Staubli VAL3: IO.dtx

public aio aAio{}
  [In4_a7CurPosH] = {link=ModbusSrv-0\Modbus-Word\In4_a7CurPosH}
  [In4_a7CurPosL] = {link=ModbusSrv-0\Modbus-Word\In4_a7CurPosL}
  [In4_a8CurPosH] = {link=ModbusSrv-0\Modbus-Word\In4_a8CurPosH}
  [In4_a8CurPosL] = {link=ModbusSrv-0\Modbus-Word\In4_a8CurPosL}
  [In_aVersion] = {link=ModbusSrv-0\Modbus-Word\In_aVersion}
  [O1_aAirPress] = {link=ModbusSrv-0\Modbus-Word\O1_aAirPress}
  [O1_aFPWM] = {link=ModbusSrv-0\Modbus-Word\O1_aFPWM}
  [O1_aLasPwr] = {link=ModbusSrv-0\Modbus-Word\O1_aLasPwr}
  [O1_aPMW] = {link=ModbusSrv-0\Modbus-Word\O1_aPMW}
  [O2_aFollowSensitive] = {link=ModbusSrv-0\Modbus-Word\O2_aFollowSensitive}
  [O2_aNull] = {link=ModbusSrv-0\Modbus-Word\O2_aNull}
  [O4_a7AiHomeH] = {link=ModbusSrv-0\Modbus-Word\O4_a7AiHomeH}
  [O4_a7AiHomeL] = {link=ModbusSrv-0\Modbus-Word\O4_a7AiHomeL}
  [O4_a7JogVelo] = {link=ModbusSrv-0\Modbus-Word\O4_a7JogVelo}
  [O4_a7MoveDis] = {link=ModbusSrv-0\Modbus-Word\O4_a7MoveDis}
  [O4_a7MovePosH] = {link=ModbusSrv-0\Modbus-Word\O4_a7MovePosH}
  [O4_a7MovePosL] = {link=ModbusSrv-0\Modbus-Word\O4_a7MovePosL}
  [O4_a7Velocity] = {link=ModbusSrv-0\Modbus-Word\O4_a7Velocity}
  [O4_a8AiHomeH] = {link=ModbusSrv-0\Modbus-Word\O4_a8AiHomeH}
  [O4_a8AiHomeL] = {link=ModbusSrv-0\Modbus-Word\O4_a8AiHomeL}
  [O4_a8JogVelo] = {link=ModbusSrv-0\Modbus-Word\O4_a8JogVelo}
  [O4_a8MoveDis] = {link=ModbusSrv-0\Modbus-Word\O4_a8MoveDis}
  [O4_a8MovePosH] = {link=ModbusSrv-0\Modbus-Word\O4_a8MovePosH}
  [O4_a8MovePosL] = {link=ModbusSrv-0\Modbus-Word\O4_a8MovePosL}
  [O4_a8Velocity] = {link=ModbusSrv-0\Modbus-Word\O4_a8Velocity}
  [Out_a114_129] = {link=ModbusSrv-0\Modbus-Word\Out_a114_129}
  [Out_a130_133] = {link=ModbusSrv-0\Modbus-Word\Out_a130_133}
  [Out_a66_81] = {link=ModbusSrv-0\Modbus-Word\Out_a66_81}
  [Out_a82_97] = {link=ModbusSrv-0\Modbus-Word\Out_a82_97}
  [Out_a98_113] = {link=ModbusSrv-0\Modbus-Word\Out_a98_113}
public bool bAxisDoorEnable
bool bDigFollowHight
public bool bDigtal[167]
  [0] = true
  [1] = true
  [2] = true
  [3] = true
  [4] = true
  [5] = true
  [6] = true
  [7] = true
  [8] = true
  [9] = true
  [10] = true
  [11] = true
  [12] = true
  [13] = true
  [14] = true
  [15] = true
  [16] = true
  [17] = true
  [18] = true
  [19] = true
  [20] = true
  [21] = true
  [22] = true
  [23] = true
  [24] = true
  [25] = true
  [26] = true
  [27] = true
  [28] = true
  [29] = true
  [30] = true
  [31] = true
  [32] = true
  [33] = true
  [34] = true
  [35] = true
  [36] = true
  [37] = true
  [38] = true
  [39] = true
  [40] = true
  [41] = true
  [42] = true
  [43] = true
  [44] = true
  [45] = true
  [46] = true
  [47] = true
  [48] = true
  [49] = true
  [50] = true
  [51] = true
  [52] = true
  [53] = true
  [54] = true
  [55] = true
  [56] = true
  [57] = true
  [58] = true
  [59] = true
  [60] = true
  [61] = true
  [62] = true
  [63] = true
  [64] = true
  [65] = true
  [66] = true
  [67] = true
  [68] = true
  [69] = true
  [70] = true
  [71] = true
  [72] = true
  [73] = true
  [74] = true
  [75] = true
  [76] = true
  [77] = true
  [78] = true
  [79] = true
  [80] = true
  [81] = true
  [82] = true
  [83] = true
  [84] = true
  [85] = true
  [86] = true
  [87] = true
  [88] = true
  [89] = true
  [90] = true
  [91] = true
  [92] = true
  [93] = true
  [94] = true
  [95] = true
  [96] = true
  [97] = true
  [98] = true
  [99] = true
  [100] = true
  [101] = true
  [102] = true
  [103] = true
  [104] = true
  [105] = true
  [106] = true
  [107] = true
  [108] = true
  [109] = true
  [110] = true
  [111] = true
  [112] = true
  [113] = true
  [114] = true
  [115] = true
  [116] = true
  [117] = true
  [118] = true
  [119] = true
  [120] = true
  [121] = true
  [122] = true
  [123] = true
  [124] = true
  [125] = true
  [126] = true
  [127] = true
  [128] = true
  [129] = true
  [130] = true
  [131] = true
  [132] = true
  [133] = true
  [134] = true
public bool bExt7AxisEnable
public bool bExt8AxisEnable
public bool bGunUp
bool bWaitActionOff
bool bWaitFollowDown
public bool bWeldEnable
public dio dDio{}
  [In1_bEndCycl] = {link=ModbusSrv-0\Modbus-Bit\In1_bEndCycl}
  [In1_bHome] = {link=ModbusSrv-0\Modbus-Bit\In1_bHome}
  [In1_bNull1] = {link=ModbusSrv-0\Modbus-Bit\In1_bNull1}
  [In1_bNull2] = {link=ModbusSrv-0\Modbus-Bit\In1_bNull2}
  [In1_bNull3] = {link=ModbusSrv-0\Modbus-Bit\In1_bNull3}
  [In1_bOutAlarm] = {link=ModbusSrv-0\Modbus-Bit\In1_bOutAlarm}
  [In1_bPausCycl] = {link=ModbusSrv-0\Modbus-Bit\In1_bPausCycl}
  [In1_bPeripheralReady] = {link=ModbusSrv-0\Modbus-Bit\In1_bPeripheralReady}
  [In1_bPowerOn] = {link=ModbusSrv-0\Modbus-Bit\In1_bPowerOn}
  [In1_bPrdSta1] = {link=ModbusSrv-0\Modbus-Bit\In1_bPrdSta1}
  [In1_bPrdSta2] = {link=ModbusSrv-0\Modbus-Bit\In1_bPrdSta2}
  [In1_bReset] = {link=ModbusSrv-0\Modbus-Bit\In1_bReset}
  [In1_bStartCycl] = {link=ModbusSrv-0\Modbus-Bit\In1_bStartCycl}
  [In1_bStopCycl] = {link=ModbusSrv-0\Modbus-Bit\In1_bStopCycl}
  [In2_bAirAlarm] = {link=ModbusSrv-0\Modbus-Bit\In2_bAirAlarm}
  [In2_bCollisonAlarm] = {link=ModbusSrv-0\Modbus-Bit\In2_bCollisonAlarm}
  [In2_bContactAlarm] = {link=ModbusSrv-0\Modbus-Bit\In2_bContactAlarm}
  [In2_bLaserAlarm] = {link=ModbusSrv-0\Modbus-Bit\In2_bLaserAlarm}
  [In2_bNull1] = {link=ModbusSrv-0\Modbus-Bit\In2_bNull1}
  [In2_bNull2] = {link=ModbusSrv-0\Modbus-Bit\In2_bNull2}
  [In2_bNull3] = {link=ModbusSrv-0\Modbus-Bit\In2_bNull3}
  [In2_bNull4] = {link=ModbusSrv-0\Modbus-Bit\In2_bNull4}
  [In2_bNull5] = {link=ModbusSrv-0\Modbus-Bit\In2_bNull5}
  [In2_bNull6] = {link=ModbusSrv-0\Modbus-Bit\In2_bNull6}
  [In2_bNull7] = {link=ModbusSrv-0\Modbus-Bit\In2_bNull7}
  [In2_bNull8] = {link=ModbusSrv-0\Modbus-Bit\In2_bNull8}
  [In2_bNull9] = {link=ModbusSrv-0\Modbus-Bit\In2_bNull9}
  [In2_bPrdSta3] = {link=ModbusSrv-0\Modbus-Bit\In2_bPrdSta3}
  [In2_bPrdSta4] = {link=ModbusSrv-0\Modbus-Bit\In2_bPrdSta4}
  [In2_bRasterOn] = {link=ModbusSrv-0\Modbus-Bit\In2_bRasterOn}
  [In4_b7BackHome] = {link=ModbusSrv-0\Modbus-Bit\In4_b7BackHome}
  [In4_b7HomeDone] = {link=ModbusSrv-0\Modbus-Bit\In4_b7HomeDone}
  [In4_b7IsHome] = {link=ModbusSrv-0\Modbus-Bit\In4_b7IsHome}
  [In4_b7MotorError] = {link=ModbusSrv-0\Modbus-Bit\In4_b7MotorError}
  [In4_b7MotorPower] = {link=ModbusSrv-0\Modbus-Bit\In4_b7MotorPower}
  [In4_b7Reached] = {link=ModbusSrv-0\Modbus-Bit\In4_b7Reached}
  [In4_b8BackHome] = {link=ModbusSrv-0\Modbus-Bit\In4_b8BackHome}
  [In4_b8HomeDone] = {link=ModbusSrv-0\Modbus-Bit\In4_b8HomeDone}
  [In4_b8IsHome] = {link=ModbusSrv-0\Modbus-Bit\In4_b8IsHome}
  [In4_b8MotorError] = {link=ModbusSrv-0\Modbus-Bit\In4_b8MotorError}
  [In4_b8MotorPower] = {link=ModbusSrv-0\Modbus-Bit\In4_b8MotorPower}
  [In4_b8Reached] = {link=ModbusSrv-0\Modbus-Bit\In4_b8Reached}
  [In4_bNull1] = {link=ModbusSrv-0\Modbus-Bit\In4_bNull1}
  [In4_bNull2] = {link=ModbusSrv-0\Modbus-Bit\In4_bNull2}
  [In4_bNull3] = {link=ModbusSrv-0\Modbus-Bit\In4_bNull3}
  [In4_bNull4] = {link=ModbusSrv-0\Modbus-Bit\In4_bNull4}
  [In4_bNull5] = {link=ModbusSrv-0\Modbus-Bit\In4_bNull5}
  [In4_bNull6] = {link=ModbusSrv-0\Modbus-Bit\In4_bNull6}
  [In4_bNull7] = {link=ModbusSrv-0\Modbus-Bit\In4_bNull7}
  [In4_bNull8] = {link=ModbusSrv-0\Modbus-Bit\In4_bNull8}
  [In7_bDownLimit_7] = {link=ModbusSrv-0\Modbus-Bit\In7_bDownLimit_7}
  [In7_bHomeLimit_7] = {link=ModbusSrv-0\Modbus-Bit\In7_bHomeLimit_7}
  [In7_bNull1] = {link=ModbusSrv-0\Modbus-Bit\In7_bNull1}
  [In7_bUpLimit_7] = {link=ModbusSrv-0\Modbus-Bit\In7_bUpLimit_7}
  [In8_bDownLimit_8] = {link=ModbusSrv-0\Modbus-Bit\In8_bDownLimit_8}
  [In8_bHomeLimit_8] = {link=ModbusSrv-0\Modbus-Bit\In8_bHomeLimit_8}
  [In8_bNull1] = {link=ModbusSrv-0\Modbus-Bit\In8_bNull1}
  [In8_bUpLimit_8] = {link=ModbusSrv-0\Modbus-Bit\In8_bUpLimit_8}
  [O1_bAirOn] = {link=ModbusSrv-0\Modbus-Bit\O1_bAirOn}
  [O1_bAlarm] = {link=ModbusSrv-0\Modbus-Bit\O1_bAlarm}
  [O1_bFollowDone] = {link=ModbusSrv-0\Modbus-Bit\O1_bFollowDone}
  [O1_bFollowOn] = {link=ModbusSrv-0\Modbus-Bit\O1_bFollowOn}
  [O1_bGreenLamp] = {link=ModbusSrv-0\Modbus-Bit\O1_bGreenLamp}
  [O1_bLaserOn] = {link=ModbusSrv-0\Modbus-Bit\O1_bLaserOn}
  [O1_bNull1] = {link=ModbusSrv-0\Modbus-Bit\O1_bNull1}
  [O1_bRedLamp] = {link=ModbusSrv-0\Modbus-Bit\O1_bRedLamp}
  [O1_bYellowLamp] = {link=ModbusSrv-0\Modbus-Bit\O1_bYellowLamp}
  [O2_bAxisPos1] = {link=ModbusSrv-0\Modbus-Bit\O2_bAxisPos1}
  [O2_bAxisPos2] = {link=ModbusSrv-0\Modbus-Bit\O2_bAxisPos2}
  [O2_bAxisPos3] = {link=ModbusSrv-0\Modbus-Bit\O2_bAxisPos3}
  [O2_bFollowHeigh1] = {link=ModbusSrv-0\Modbus-Bit\O2_bFollowHeigh1}
  [O2_bFollowHeigh2] = {link=ModbusSrv-0\Modbus-Bit\O2_bFollowHeigh2}
  [O2_bFollowHeigh3] = {link=ModbusSrv-0\Modbus-Bit\O2_bFollowHeigh3}
  [O2_bNull1] = {link=ModbusSrv-0\Modbus-Bit\O2_bNull1}
  [O2_bNull2] = {link=ModbusSrv-0\Modbus-Bit\O2_bNull2}
  [O2_bNull3] = {link=ModbusSrv-0\Modbus-Bit\O2_bNull3}
  [O2_bProCode1] = {link=ModbusSrv-0\Modbus-Bit\O2_bProCode1}
  [O2_bProCode2] = {link=ModbusSrv-0\Modbus-Bit\O2_bProCode2}
  [O2_bProCode3] = {link=ModbusSrv-0\Modbus-Bit\O2_bProCode3}
  [O2_bSta1Stat] = {link=ModbusSrv-0\Modbus-Bit\O2_bSta1Stat}
  [O2_bSta2Stat] = {link=ModbusSrv-0\Modbus-Bit\O2_bSta2Stat}
  [O2_bSta3Stat] = {link=ModbusSrv-0\Modbus-Bit\O2_bSta3Stat}
  [O2_bSta4Stat] = {link=ModbusSrv-0\Modbus-Bit\O2_bSta4Stat}
  [O4_b7AxisHome] = {link=ModbusSrv-0\Modbus-Bit\O4_b7AxisHome}
  [O4_b7ChkHome] = {link=ModbusSrv-0\Modbus-Bit\O4_b7ChkHome}
  [O4_b7MoveDir] = {link=ModbusSrv-0\Modbus-Bit\O4_b7MoveDir}
  [O4_b7MoveDirM] = {link=ModbusSrv-0\Modbus-Bit\O4_b7MoveDirM}
  [O4_b7MoveToPos] = {link=ModbusSrv-0\Modbus-Bit\O4_b7MoveToPos}
  [O4_b7RecordPos] = {link=ModbusSrv-0\Modbus-Bit\O4_b7RecordPos}
  [O4_b7ResetError] = {link=ModbusSrv-0\Modbus-Bit\O4_b7ResetError}
  [O4_b7StopMotor] = {link=ModbusSrv-0\Modbus-Bit\O4_b7StopMotor}
  [O4_b8AxisHome] = {link=ModbusSrv-0\Modbus-Bit\O4_b8AxisHome}
  [O4_b8ChkHome] = {link=ModbusSrv-0\Modbus-Bit\O4_b8ChkHome}
  [O4_b8MoveDir] = {link=ModbusSrv-0\Modbus-Bit\O4_b8MoveDir}
  [O4_b8MoveDirM] = {link=ModbusSrv-0\Modbus-Bit\O4_b8MoveDirM}
  [O4_b8MoveToPos] = {link=ModbusSrv-0\Modbus-Bit\O4_b8MoveToPos}
  [O4_b8RecordPos] = {link=ModbusSrv-0\Modbus-Bit\O4_b8RecordPos}
  [O4_b8ResetError] = {link=ModbusSrv-0\Modbus-Bit\O4_b8ResetError}
  [O4_b8StopMotor] = {link=ModbusSrv-0\Modbus-Bit\O4_b8StopMotor}
  [O4_bHome] = {link=ModbusSrv-0\Modbus-Bit\O4_bHome}
  [O4_bNull1] = {link=ModbusSrv-0\Modbus-Bit\O4_bNull1}
  [O4_bNull2] = {link=ModbusSrv-0\Modbus-Bit\O4_bNull2}
  [O4_bNull3] = {link=ModbusSrv-0\Modbus-Bit\O4_bNull3}
  [O4_bNull4] = {link=ModbusSrv-0\Modbus-Bit\O4_bNull4}
  [O4_bNull5] = {link=ModbusSrv-0\Modbus-Bit\O4_bNull5}
  [O4_bNull6] = {link=ModbusSrv-0\Modbus-Bit\O4_bNull6}
  [O4_bNull7] = {link=ModbusSrv-0\Modbus-Bit\O4_bNull7}
  [O4_bNull8] = {link=ModbusSrv-0\Modbus-Bit\O4_bNull8}
  [O7_bAxis7Direction] = {link=ModbusSrv-0\Modbus-Bit\O7_bAxis7Direction}
  [O7_bAxis7Pulse] = {link=ModbusSrv-0\Modbus-Bit\O7_bAxis7Pulse}
  [O7_bNull1] = {link=ModbusSrv-0\Modbus-Bit\O7_bNull1}
  [O7_bNull2] = {link=ModbusSrv-0\Modbus-Bit\O7_bNull2}
  [O7_bNull3] = {link=ModbusSrv-0\Modbus-Bit\O7_bNull3}
  [O8_bAxis8Direction] = {link=ModbusSrv-0\Modbus-Bit\O8_bAxis8Direction}
  [O8_bAxis8Pulse] = {link=ModbusSrv-0\Modbus-Bit\O8_bAxis8Pulse}
  [O8_bNull1] = {link=ModbusSrv-0\Modbus-Bit\O8_bNull1}
  [O8_bNull2] = {link=ModbusSrv-0\Modbus-Bit\O8_bNull2}
  [O8_bNull3] = {link=ModbusSrv-0\Modbus-Bit\O8_bNull3}
  [UsIn_bNull1] = {link=ModbusSrv-0\Modbus-Bit\UsIn_bNull1}
  [UsIn_bNull2] = {link=ModbusSrv-0\Modbus-Bit\UsIn_bNull2}
  [UsIn_bNull3] = {link=ModbusSrv-0\Modbus-Bit\UsIn_bNull3}
  [UsIn_bNull4] = {link=ModbusSrv-0\Modbus-Bit\UsIn_bNull4}
  [UsIn_bNull5] = {link=ModbusSrv-0\Modbus-Bit\UsIn_bNull5}
  [UsIn_bNull6] = {link=ModbusSrv-0\Modbus-Bit\UsIn_bNull6}
  [UsIn_bNull7] = {link=ModbusSrv-0\Modbus-Bit\UsIn_bNull7}
  [UsIn_bNull8] = {link=ModbusSrv-0\Modbus-Bit\UsIn_bNull8}
  [UsO_bNull1] = {link=ModbusSrv-0\Modbus-Bit\UsO_bNull1}
  [UsO_bNull2] = {link=ModbusSrv-0\Modbus-Bit\UsO_bNull2}
  [UsO_bNull3] = {link=ModbusSrv-0\Modbus-Bit\UsO_bNull3}
  [UsO_bNull4] = {link=ModbusSrv-0\Modbus-Bit\UsO_bNull4}
  [UsO_bNull5] = {link=ModbusSrv-0\Modbus-Bit\UsO_bNull5}
  [UsO_bNull6] = {link=ModbusSrv-0\Modbus-Bit\UsO_bNull6}
  [UsO_bNull7] = {link=ModbusSrv-0\Modbus-Bit\UsO_bNull7}
  [UsO_bNull8] = {link=ModbusSrv-0\Modbus-Bit\UsO_bNull8}
public string sIOName[167]
  [0] = "无"
  [1] = "In1_bPowerOn"
  [2] = "In1_bStartCycl"
  [3] = "In1_bStopCycl"
  [4] = "In1_bHome"
  [5] = "In1_bEndCycl"
  [6] = "In1_bPrdSta1"
  [7] = "In1_bPrdSta2"
  [8] = "In1_bPausCycl"
  [9] = "In1_bOutAlarm"
  [10] = "In1_bReset"
  [11] = "In1_bPeripheralReady"
  [12] = "In1_bNull1"
  [13] = "In1_bNull2"
  [14] = "In1_bNull3"
  [15] = "UsIn_bNull1"
  [16] = "UsIn_bNull2"
  [17] = "UsIn_bNull3"
  [18] = "UsIn_bNull4"
  [19] = "UsIn_bNull5"
  [20] = "UsIn_bNull6"
  [21] = "UsIn_bNull7"
  [22] = "UsIn_bNull8"
  [23] = "In2_bPrdSta3"
  [24] = "In2_bPrdSta4"
  [25] = "In2_bAirAlarm"
  [26] = "In2_bCollisonAlarm"
  [27] = "In2_bLaserAlarm"
  [28] = "In2_bContactAlarm"
  [29] = "In2_bRasterOn"
  [30] = "In2_bNull1"
  [31] = "In2_bNull2"
  [32] = "In2_bNull3"
  [33] = "In2_bNull4"
  [34] = "In2_bNull5"
  [35] = "In2_bNull6"
  [36] = "In2_bNull7"
  [37] = "In2_bNull8"
  [38] = "In2_bNull9"
  [39] = "In7_bUpLimit_7"
  [40] = "In7_bDownLimit_7"
  [41] = "In7_bHomeLimit_7"
  [42] = "In7_bNull1"
  [43] = "In8_bUpLimit_8"
  [44] = "In8_bDownLimit_8"
  [45] = "In8_bHomeLimit_8"
  [46] = "In8_bNull1"
  [47] = "In4_b7Reached"
  [48] = "In4_b7BackHome"
  [49] = "In4_b7HomeDone"
  [50] = "In4_b7MotorPower"
  [51] = "In4_b7IsHome"
  [52] = "In4_b7MotorError"
  [53] = "In4_b8Reached"
  [54] = "In4_b8BackHome"
  [55] = "In4_b8HomeDone"
  [56] = "In4_b8MotorPower"
  [57] = "In4_b8IsHome"
  [58] = "In4_b8MotorError"
  [59] = "In4_bNull1"
  [60] = "In4_bNull2"
  [61] = "In4_bNull3"
  [62] = "In4_bNull4"
  [63] = "In4_bNull5"
  [64] = "In4_bNull6"
  [65] = "In4_bNull7"
  [66] = "In4_bNull8"
  [67] = "O1_bLaserOn"
  [68] = "O1_bFollowOn"
  [69] = "O1_bFollowDone"
  [70] = "O1_bAirOn"
  [71] = "O1_bNull1"
  [72] = "O1_bRedLamp"
  [73] = "O1_bYellowLamp"
  [74] = "O1_bGreenLamp"
  [75] = "O1_bAlarm"
  [76] = "UsO_bNull1"
  [77] = "UsO_bNull2"
  [78] = "UsO_bNull3"
  [79] = "UsO_bNull4"
  [80] = "UsO_bNull5"
  [81] = "UsO_bNull6"
  [82] = "UsO_bNull7"
  [83] = "UsO_bNull8"
  [84] = "O2_bSta1Stat"
  [85] = "O2_bSta2Stat"
  [86] = "O2_bSta3Stat"
  [87] = "O2_bSta4Stat"
  [88] = "O2_bProCode1"
  [89] = "O2_bProCode2"
  [90] = "O2_bProCode3"
  [91] = "O2_bFollowHeigh1"
  [92] = "O2_bFollowHeigh2"
  [93] = "O2_bFollowHeigh3"
  [94] = "O2_bAxisPos1"
  [95] = "O2_bAxisPos2"
  [96] = "O2_bAxisPos3"
  [97] = "O2_bNull1"
  [98] = "O2_bNull2"
  [99] = "O2_bNull3"
  [100] = "O7_bAxis7Pulse"
  [101] = "O7_bAxis7Direction"
  [102] = "O7_bNull1"
  [103] = "O7_bNull2"
  [104] = "O7_bNull3"
  [105] = "O8_bAxis8Pulse"
  [106] = "O8_bAxis8Direction"
  [107] = "O8_bNull1"
  [108] = "O8_bNull2"
  [109] = "O8_bNull3"
  [110] = "O4_b7RecordPos"
  [111] = "O4_b7MoveToPos"
  [112] = "O4_b7ResetError"
  [113] = "O4_b7ChkHome"
  [114] = "O4_b7AxisHome"
  [115] = "O4_b7MoveDir"
  [116] = "O4_b7MoveDirM"
  [117] = "O4_b7StopMotor"
  [118] = "O4_bHome"
  [119] = "O4_b8RecordPos"
  [120] = "O4_b8MoveToPos"
  [121] = "O4_b8ResetError"
  [122] = "O4_b8ChkHome"
  [123] = "O4_b8AxisHome"
  [124] = "O4_b8MoveDir"
  [125] = "O4_b8MoveDirM"
  [126] = "O4_b8StopMotor"
  [127] = "O4_bNull1"
  [128] = "O4_bNull2"
  [129] = "O4_bNull3"
  [130] = "O4_bNull4"
  [131] = "O4_bNull5"
  [132] = "O4_bNull6"
  [133] = "O4_bNull7"
  [134] = "O4_bNull8"
  [135] = "O1_aLasPwr"
  [136] = "O1_aAirPress"
  [137] = "O1_aFPWM"
  [138] = "O1_aPMW"
  [139] = "O2_aFollowSensitive"
  [140] = "O2_aNull"
  [141] = "In4_a7CurPosL"
  [142] = "In4_a7CurPosH"
  [143] = "In4_a8CurPosL"
  [144] = "In4_a8CurPosH"
  [145] = "O4_a7Velocity"
  [146] = "O4_a7JogVelo"
  [147] = "O4_a7MoveDis"
  [148] = "O4_a7AiHomeH"
  [149] = "O4_a7AiHomeL"
  [150] = "O4_a7MovePosL"
  [151] = "O4_a7MovePosH"
  [152] = "O4_a8Velocity"
  [153] = "O4_a8JogVelo"
  [154] = "O4_a8MoveDis"
  [155] = "O4_a8AiHomeH"
  [156] = "O4_a8AiHomeL"
  [157] = "O4_a8MovePosL"
  [158] = "O4_a8MovePosH"
  [159] = "Out_a66_81"
  [160] = "Out_a82_97"
  [161] = "Out_a98_113"
  [162] = "Out_a114_129"
  [163] = "Out_a130_133"
  [164] = "In_aVersion"
  [165] = "延时"
  [166] = "收弧时间"
public bool bUserIOReset
